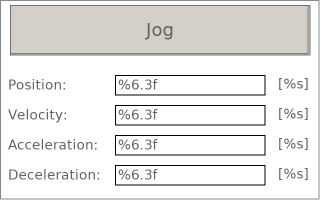
VISUALIZATION SingleAxisJogInchingModulo  // 320x200
VAR_IN_OUT
	btnJogPositive	: BOOL;
	btnJogNegative	: BOOL;
	lrPosition		: LREAL;
	lrVelocity		: LREAL;
	lrAcceleration	: LREAL;
	lrDeceleration	: LREAL;
	sUnit			: STRING;
END_VAR
    Rectangle (5,75 110x20), "Position:"
    Rectangle (115,75 150x20), "%6.3f", text variable: lrPosition
        OnMouseClick: write the text variable via VisuDialogs.Numpad
    Rectangle (275,75 44x18), "[%s]", text variable: sUnit
    Button (10,5 300x50), "Jog"
        tap btnJogPositive
    Rectangle (5,105 110x20), "Velocity:"
    Rectangle (115,105 150x20), "%6.3f", text variable: lrVelocity
        OnMouseClick: write the text variable via VisuDialogs.Numpad
    Rectangle (275,105 44x18), "[%s]", text variable: sUnit
    Rectangle (5,135 110x20), "Acceleration:"
    Rectangle (115,135 150x20), "%6.3f", text variable: lrAcceleration
        OnMouseClick: write the text variable via VisuDialogs.Numpad
    Rectangle (275,135 44x18), "[%s]", text variable: sUnit
    Rectangle (5,165 110x20), "Deceleration:"
    Rectangle (115,165 150x20), "%6.3f", text variable: lrDeceleration
        OnMouseClick: write the text variable via VisuDialogs.Numpad
    Rectangle (275,165 44x18), "[%s]", text variable: sUnit
END_VISUALIZATION

(* stored: Version 1.1.0.1, ProductVersion 3.1.4024.9
   Visu SingleAxisJogInchingModulo: Id {e99f2d53-57eb-4ba6-98d3-95e146688fba} *)
